KUKA KRL program: PROTON_EXHIBITION.src, PROTON_EXHIBITION.dat

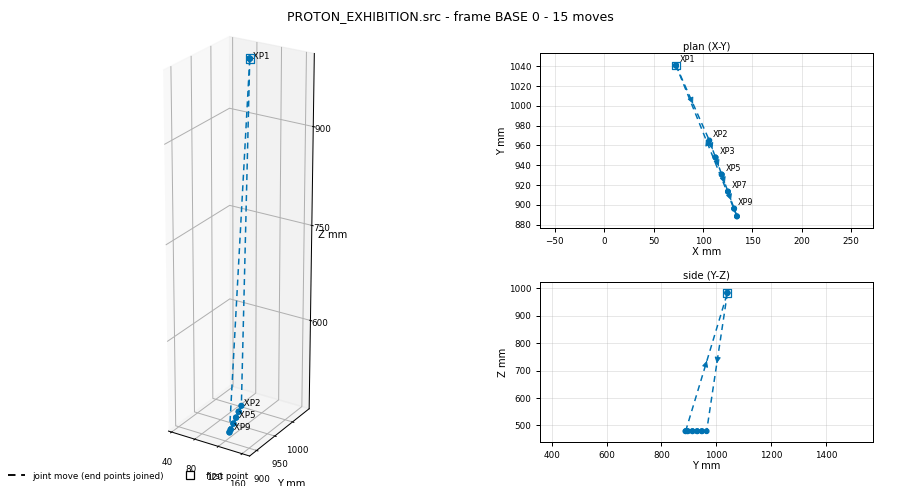
[picture p0: tool path of PROTON_EXHIBITION.src in frame BASE 0, 15 of 15 moves have a stored position in this frame; points joined in program order, loops and branches not executed]
--- PROTON_EXHIBITION.src ---
&ACCESS RVP
&REL 2
&PARAM DISKPATH = KRC:\\R1\\Program
DEF PROTON_EXHIBITION()
   DECL INT RET
   DECL INT CMD
   DECL REAL OUT_PULSE_TIME

   BAS(#INITMOV, 0)
   CMD = 0
   OUT_PULSE_TIME = 1.0

   \
       ;FOLD SPTP P1 Vel=100 % PDAT1 Tool[1]:Tool Base[0] ;%{PE}
       ;FOLD Parameters ;%{h}
       ;Params IlfProvider=kukaroboter.basistech.inlineforms.movement.spline; Kuka.IsGlobalPoint=False; Kuka.PointName=P1; Kuka.BlendingEnabled=False; Kuka.MoveDataPtpName=PDAT1; Kuka.VelocityPtp=100; Kuka.VelocityFieldEnabled=True; Kuka.ColDetectFieldEnabled=True; Kuka.CurrentCDSetIndex=0; Kuka.MovementParameterFieldEnabled=True; IlfCommand=SPTP
       ;ENDFOLD
       SPTP XP1 WITH $VEL_AXIS[1] = SVEL_JOINT(100.0), $TOOL = STOOL2(FP1), $BASE = SBASE(FP1.BASE_NO), $IPO_MODE = SIPO_MODE(FP1.IPO_FRAME), $LOAD = SLOAD(FP1.TOOL_NO), $ACC_AXIS[1] = SACC_JOINT(PPDAT1), $APO = SAPO_PTP(PPDAT1), $GEAR_JERK[1] = SGEAR_JERK(PPDAT1), $COLLMON_TOL_PRO[1] = USE_CM_PRO_VALUES(0)
       ;ENDFOLD

   LOOP
      ; ready to start = 0
      RET = EKI_SetInt("STATUS_EKI", "Status", 0)
      RET = EKI_Send("STATUS_EKI")

      ; wait for start cycle command, expected Cmd = 1
      CMD = 0
      REPEAT
         WAIT SEC 0.05
         RET = EKI_ReadNext("STATUS_EKI")
         IF RET == EkiOk THEN
            RET = EKI_GetInt("STATUS_EKI", "Cmd", CMD)
         ENDIF
      UNTIL (RET == EkiOk) AND (CMD == 1)

      ; next_position = 1
      RET = EKI_SetInt("STATUS_EKI", "Status", 1)
      RET = EKI_Send("STATUS_EKI")

   \
       ;FOLD SPTP P1 Vel=100 % PDAT1 Tool[1]:Tool Base[0] ;%{PE}
       ;FOLD Parameters ;%{h}
       ;Params IlfProvider=kukaroboter.basistech.inlineforms.movement.spline; Kuka.IsGlobalPoint=False; Kuka.PointName=P1; Kuka.BlendingEnabled=False; Kuka.MoveDataPtpName=PDAT1; Kuka.VelocityPtp=100; Kuka.VelocityFieldEnabled=True; Kuka.ColDetectFieldEnabled=True; Kuka.CurrentCDSetIndex=0; Kuka.MovementParameterFieldEnabled=True; IlfCommand=SPTP
       ;ENDFOLD
       SPTP XP1 WITH $VEL_AXIS[1] = SVEL_JOINT(100.0), $TOOL = STOOL2(FP1), $BASE = SBASE(FP1.BASE_NO), $IPO_MODE = SIPO_MODE(FP1.IPO_FRAME), $LOAD = SLOAD(FP1.TOOL_NO), $ACC_AXIS[1] = SACC_JOINT(PPDAT1), $APO = SAPO_PTP(PPDAT1), $GEAR_JERK[1] = SGEAR_JERK(PPDAT1), $COLLMON_TOL_PRO[1] = USE_CM_PRO_VALUES(0)
       ;ENDFOLD

      ; in_position = 2
      WAIT FOR $OUT[1] == FALSE
      RET = EKI_SetInt("STATUS_EKI", "Status", 2)
      RET = EKI_Send("STATUS_EKI")

      ; wait command to move to P2
      CMD = 0
      REPEAT
         WAIT SEC 0.05
         RET = EKI_ReadNext("STATUS_EKI")
         IF RET == EkiOk THEN
            RET = EKI_GetInt("STATUS_EKI", "Cmd", CMD)
         ENDIF
      UNTIL (RET == EkiOk) AND (CMD == 1)

      ; next_position = 1
      RET = EKI_SetInt("STATUS_EKI", "Status", 1)
      RET = EKI_Send("STATUS_EKI")
      PULSE($OUT[1], TRUE, OUT_PULSE_TIME)

      \
          ;FOLD SPTP P2 Vel=100 % PDAT2 Tool[1]:Tool Base[0] ;%{PE}
          ;FOLD Parameters ;%{h}
          ;Params IlfProvider=kukaroboter.basistech.inlineforms.movement.spline; Kuka.IsGlobalPoint=False; Kuka.PointName=P2; Kuka.BlendingEnabled=False; Kuka.MoveDataPtpName=PDAT2; Kuka.VelocityPtp=100; Kuka.VelocityFieldEnabled=True; Kuka.ColDetectFieldEnabled=True; Kuka.CurrentCDSetIndex=0; Kuka.MovementParameterFieldEnabled=True; IlfCommand=SPTP
          ;ENDFOLD
          SPTP XP2 WITH $VEL_AXIS[1] = SVEL_JOINT(100.0), $TOOL = STOOL2(FP2), $BASE = SBASE(FP2.BASE_NO), $IPO_MODE = SIPO_MODE(FP2.IPO_FRAME), $LOAD = SLOAD(FP2.TOOL_NO), $ACC_AXIS[1] = SACC_JOINT(PPDAT2), $APO = SAPO_PTP(PPDAT2), $GEAR_JERK[1] = SGEAR_JERK(PPDAT2), $COLLMON_TOL_PRO[1] = USE_CM_PRO_VALUES(0)
          ;ENDFOLD

      ; in_position = 2
      WAIT FOR $OUT[1] == FALSE
      RET = EKI_SetInt("STATUS_EKI", "Status", 2)
      RET = EKI_Send("STATUS_EKI")

      ; wait command to move to P3
      CMD = 0
      REPEAT
         WAIT SEC 0.05
         RET = EKI_ReadNext("STATUS_EKI")
         IF RET == EkiOk THEN
            RET = EKI_GetInt("STATUS_EKI", "Cmd", CMD)
         ENDIF
      UNTIL (RET == EkiOk) AND (CMD == 1)

      ; next_position = 1
      RET = EKI_SetInt("STATUS_EKI", "Status", 1)
      RET = EKI_Send("STATUS_EKI")
      PULSE($OUT[1], TRUE, OUT_PULSE_TIME)

      \
          ;FOLD SPTP P3 Vel=100 % PDAT3 Tool[1]:Tool Base[0] ;%{PE}
          ;FOLD Parameters ;%{h}
          ;Params IlfProvider=kukaroboter.basistech.inlineforms.movement.spline; Kuka.IsGlobalPoint=False; Kuka.PointName=P3; Kuka.BlendingEnabled=False; Kuka.MoveDataPtpName=PDAT3; Kuka.VelocityPtp=100; Kuka.VelocityFieldEnabled=True; Kuka.ColDetectFieldEnabled=True; Kuka.CurrentCDSetIndex=0; Kuka.MovementParameterFieldEnabled=True; IlfCommand=SPTP
          ;ENDFOLD
          SPTP XP3 WITH $VEL_AXIS[1] = SVEL_JOINT(100.0), $TOOL = STOOL2(FP3), $BASE = SBASE(FP3.BASE_NO), $IPO_MODE = SIPO_MODE(FP3.IPO_FRAME), $LOAD = SLOAD(FP3.TOOL_NO), $ACC_AXIS[1] = SACC_JOINT(PPDAT3), $APO = SAPO_PTP(PPDAT3), $GEAR_JERK[1] = SGEAR_JERK(PPDAT3), $COLLMON_TOL_PRO[1] = USE_CM_PRO_VALUES(0)
          ;ENDFOLD

      ; in_position = 2
      WAIT FOR $OUT[1] == FALSE
      RET = EKI_SetInt("STATUS_EKI", "Status", 2)
      RET = EKI_Send("STATUS_EKI")

      ; wait command to move to P4
      CMD = 0
      REPEAT
         WAIT SEC 0.05
         RET = EKI_ReadNext("STATUS_EKI")
         IF RET == EkiOk THEN
            RET = EKI_GetInt("STATUS_EKI", "Cmd", CMD)
         ENDIF
      UNTIL (RET == EkiOk) AND (CMD == 1)

      ; next_position = 1
      RET = EKI_SetInt("STATUS_EKI", "Status", 1)
      RET = EKI_Send("STATUS_EKI")
      PULSE($OUT[1], TRUE, OUT_PULSE_TIME)

      \
          ;FOLD SPTP P4 Vel=100 % PDAT4 Tool[1]:Tool Base[0] ;%{PE}
          ;FOLD Parameters ;%{h}
          ;Params IlfProvider=kukaroboter.basistech.inlineforms.movement.spline; Kuka.IsGlobalPoint=False; Kuka.PointName=P4; Kuka.BlendingEnabled=False; Kuka.MoveDataPtpName=PDAT4; Kuka.VelocityPtp=100; Kuka.VelocityFieldEnabled=True; Kuka.ColDetectFieldEnabled=True; Kuka.CurrentCDSetIndex=0; Kuka.MovementParameterFieldEnabled=True; IlfCommand=SPTP
          ;ENDFOLD
          SPTP XP4 WITH $VEL_AXIS[1] = SVEL_JOINT(100.0), $TOOL = STOOL2(FP4), $BASE = SBASE(FP4.BASE_NO), $IPO_MODE = SIPO_MODE(FP4.IPO_FRAME), $LOAD = SLOAD(FP4.TOOL_NO), $ACC_AXIS[1] = SACC_JOINT(PPDAT4), $APO = SAPO_PTP(PPDAT4), $GEAR_JERK[1] = SGEAR_JERK(PPDAT4), $COLLMON_TOL_PRO[1] = USE_CM_PRO_VALUES(0)
          ;ENDFOLD

      ; in_position = 2
      WAIT FOR $OUT[1] == FALSE
      RET = EKI_SetInt("STATUS_EKI", "Status", 2)
      RET = EKI_Send("STATUS_EKI")

      ; wait command to move to P5
      CMD = 0
      REPEAT
         WAIT SEC 0.05
         RET = EKI_ReadNext("STATUS_EKI")
         IF RET == EkiOk THEN
            RET = EKI_GetInt("STATUS_EKI", "Cmd", CMD)
         ENDIF
      UNTIL (RET == EkiOk) AND (CMD == 1)

      ; next_position = 1
      RET = EKI_SetInt("STATUS_EKI", "Status", 1)
      RET = EKI_Send("STATUS_EKI")
      PULSE($OUT[1], TRUE, OUT_PULSE_TIME)

      \
          ;FOLD SPTP P5 Vel=100 % PDAT5 Tool[1]:Tool Base[0] ;%{PE}
          ;FOLD Parameters ;%{h}
          ;Params IlfProvider=kukaroboter.basistech.inlineforms.movement.spline; Kuka.IsGlobalPoint=False; Kuka.PointName=P5; Kuka.BlendingEnabled=False; Kuka.MoveDataPtpName=PDAT5; Kuka.VelocityPtp=100; Kuka.VelocityFieldEnabled=True; Kuka.ColDetectFieldEnabled=True; Kuka.CurrentCDSetIndex=0; Kuka.MovementParameterFieldEnabled=True; IlfCommand=SPTP
          ;ENDFOLD
          SPTP XP5 WITH $VEL_AXIS[1] = SVEL_JOINT(100.0), $TOOL = STOOL2(FP5), $BASE = SBASE(FP5.BASE_NO), $IPO_MODE = SIPO_MODE(FP5.IPO_FRAME), $LOAD = SLOAD(FP5.TOOL_NO), $ACC_AXIS[1] = SACC_JOINT(PPDAT5), $APO = SAPO_PTP(PPDAT5), $GEAR_JERK[1] = SGEAR_JERK(PPDAT5), $COLLMON_TOL_PRO[1] = USE_CM_PRO_VALUES(0)
          ;ENDFOLD

      ; in_position = 2
      WAIT FOR $OUT[1] == FALSE
      RET = EKI_SetInt("STATUS_EKI", "Status", 2)
      RET = EKI_Send("STATUS_EKI")

      ; wait command to move to P6
      CMD = 0
      REPEAT
         WAIT SEC 0.05
         RET = EKI_ReadNext("STATUS_EKI")
         IF RET == EkiOk THEN
            RET = EKI_GetInt("STATUS_EKI", "Cmd", CMD)
         ENDIF
      UNTIL (RET == EkiOk) AND (CMD == 1)

      ; next_position = 1
      RET = EKI_SetInt("STATUS_EKI", "Status", 1)
      RET = EKI_Send("STATUS_EKI")
      PULSE($OUT[1], TRUE, OUT_PULSE_TIME)

      \
          ;FOLD SPTP P6 Vel=100 % PDAT6 Tool[1]:Tool Base[0] ;%{PE}
          ;FOLD Parameters ;%{h}
          ;Params IlfProvider=kukaroboter.basistech.inlineforms.movement.spline; Kuka.IsGlobalPoint=False; Kuka.PointName=P6; Kuka.BlendingEnabled=False; Kuka.MoveDataPtpName=PDAT6; Kuka.VelocityPtp=100; Kuka.VelocityFieldEnabled=True; Kuka.ColDetectFieldEnabled=True; Kuka.CurrentCDSetIndex=0; Kuka.MovementParameterFieldEnabled=True; IlfCommand=SPTP
          ;ENDFOLD
          SPTP XP6 WITH $VEL_AXIS[1] = SVEL_JOINT(100.0), $TOOL = STOOL2(FP6), $BASE = SBASE(FP6.BASE_NO), $IPO_MODE = SIPO_MODE(FP6.IPO_FRAME), $LOAD = SLOAD(FP6.TOOL_NO), $ACC_AXIS[1] = SACC_JOINT(PPDAT6), $APO = SAPO_PTP(PPDAT6), $GEAR_JERK[1] = SGEAR_JERK(PPDAT6), $COLLMON_TOL_PRO[1] = USE_CM_PRO_VALUES(0)
          ;ENDFOLD

      ; in_position = 2
      WAIT FOR $OUT[1] == FALSE
      RET = EKI_SetInt("STATUS_EKI", "Status", 2)
      RET = EKI_Send("STATUS_EKI")

      ; wait command to move to P7
      CMD = 0
      REPEAT
         WAIT SEC 0.05
         RET = EKI_ReadNext("STATUS_EKI")
         IF RET == EkiOk THEN
            RET = EKI_GetInt("STATUS_EKI", "Cmd", CMD)
         ENDIF
      UNTIL (RET == EkiOk) AND (CMD == 1)

      ; next_position = 1
      RET = EKI_SetInt("STATUS_EKI", "Status", 1)
      RET = EKI_Send("STATUS_EKI")
      PULSE($OUT[1], TRUE, OUT_PULSE_TIME)

      \
          ;FOLD SPTP P7 Vel=100 % PDAT7 Tool[1]:Tool Base[0] ;%{PE}
          ;FOLD Parameters ;%{h}
          ;Params IlfProvider=kukaroboter.basistech.inlineforms.movement.spline; Kuka.IsGlobalPoint=False; Kuka.PointName=P7; Kuka.BlendingEnabled=False; Kuka.MoveDataPtpName=PDAT7; Kuka.VelocityPtp=100; Kuka.VelocityFieldEnabled=True; Kuka.ColDetectFieldEnabled=True; Kuka.CurrentCDSetIndex=0; Kuka.MovementParameterFieldEnabled=True; IlfCommand=SPTP
          ;ENDFOLD
          SPTP XP7 WITH $VEL_AXIS[1] = SVEL_JOINT(100.0), $TOOL = STOOL2(FP7), $BASE = SBASE(FP7.BASE_NO), $IPO_MODE = SIPO_MODE(FP7.IPO_FRAME), $LOAD = SLOAD(FP7.TOOL_NO), $ACC_AXIS[1] = SACC_JOINT(PPDAT7), $APO = SAPO_PTP(PPDAT7), $GEAR_JERK[1] = SGEAR_JERK(PPDAT7), $COLLMON_TOL_PRO[1] = USE_CM_PRO_VALUES(0)
          ;ENDFOLD

      ; in_position = 2
      WAIT FOR $OUT[1] == FALSE
      RET = EKI_SetInt("STATUS_EKI", "Status", 2)
      RET = EKI_Send("STATUS_EKI")

      ; wait command to move to P8
      CMD = 0
      REPEAT
         WAIT SEC 0.05
         RET = EKI_ReadNext("STATUS_EKI")
         IF RET == EkiOk THEN
            RET = EKI_GetInt("STATUS_EKI", "Cmd", CMD)
         ENDIF
      UNTIL (RET == EkiOk) AND (CMD == 1)

      ; next_position = 1
      RET = EKI_SetInt("STATUS_EKI", "Status", 1)
      RET = EKI_Send("STATUS_EKI")
      PULSE($OUT[1], TRUE, OUT_PULSE_TIME)

      \
          ;FOLD SPTP P8 Vel=100 % PDAT8 Tool[1]:Tool Base[0] ;%{PE}
          ;FOLD Parameters ;%{h}
          ;Params IlfProvider=kukaroboter.basistech.inlineforms.movement.spline; Kuka.IsGlobalPoint=False; Kuka.PointName=P8; Kuka.BlendingEnabled=False; Kuka.MoveDataPtpName=PDAT8; Kuka.VelocityPtp=100; Kuka.VelocityFieldEnabled=True; Kuka.ColDetectFieldEnabled=True; Kuka.CurrentCDSetIndex=0; Kuka.MovementParameterFieldEnabled=True; IlfCommand=SPTP
          ;ENDFOLD
          SPTP XP8 WITH $VEL_AXIS[1] = SVEL_JOINT(100.0), $TOOL = STOOL2(FP8), $BASE = SBASE(FP8.BASE_NO), $IPO_MODE = SIPO_MODE(FP8.IPO_FRAME), $LOAD = SLOAD(FP8.TOOL_NO), $ACC_AXIS[1] = SACC_JOINT(PPDAT8), $APO = SAPO_PTP(PPDAT8), $GEAR_JERK[1] = SGEAR_JERK(PPDAT8), $COLLMON_TOL_PRO[1] = USE_CM_PRO_VALUES(0)
          ;ENDFOLD

      ; in_position = 2
      WAIT FOR $OUT[1] == FALSE
      RET = EKI_SetInt("STATUS_EKI", "Status", 2)
      RET = EKI_Send("STATUS_EKI")

      ; wait command to move to P9
      CMD = 0
      REPEAT
         WAIT SEC 0.05
         RET = EKI_ReadNext("STATUS_EKI")
         IF RET == EkiOk THEN
            RET = EKI_GetInt("STATUS_EKI", "Cmd", CMD)
         ENDIF
      UNTIL (RET == EkiOk) AND (CMD == 1)

      ; next_position = 1
      RET = EKI_SetInt("STATUS_EKI", "Status", 1)
      RET = EKI_Send("STATUS_EKI")
      PULSE($OUT[1], TRUE, OUT_PULSE_TIME)

      \
          ;FOLD SPTP P9 Vel=100 % PDAT9 Tool[1]:Tool Base[0] ;%{PE}
          ;FOLD Parameters ;%{h}
          ;Params IlfProvider=kukaroboter.basistech.inlineforms.movement.spline; Kuka.IsGlobalPoint=False; Kuka.PointName=P9; Kuka.BlendingEnabled=False; Kuka.MoveDataPtpName=PDAT9; Kuka.VelocityPtp=100; Kuka.VelocityFieldEnabled=True; Kuka.ColDetectFieldEnabled=True; Kuka.CurrentCDSetIndex=0; Kuka.MovementParameterFieldEnabled=True; IlfCommand=SPTP
          ;ENDFOLD
          SPTP XP9 WITH $VEL_AXIS[1] = SVEL_JOINT(100.0), $TOOL = STOOL2(FP9), $BASE = SBASE(FP9.BASE_NO), $IPO_MODE = SIPO_MODE(FP9.IPO_FRAME), $LOAD = SLOAD(FP9.TOOL_NO), $ACC_AXIS[1] = SACC_JOINT(PPDAT9), $APO = SAPO_PTP(PPDAT9), $GEAR_JERK[1] = SGEAR_JERK(PPDAT9), $COLLMON_TOL_PRO[1] = USE_CM_PRO_VALUES(0)
          ;ENDFOLD

      ; in_position = 2
      WAIT FOR $OUT[1] == FALSE
      RET = EKI_SetInt("STATUS_EKI", "Status", 2)
      RET = EKI_Send("STATUS_EKI")

      ; wait command to move to P10
      CMD = 0
      REPEAT
         WAIT SEC 0.05
         RET = EKI_ReadNext("STATUS_EKI")
         IF RET == EkiOk THEN
            RET = EKI_GetInt("STATUS_EKI", "Cmd", CMD)
         ENDIF
      UNTIL (RET == EkiOk) AND (CMD == 1)

      ; next_position = 1
      RET = EKI_SetInt("STATUS_EKI", "Status", 1)
      RET = EKI_Send("STATUS_EKI")
      PULSE($OUT[1], TRUE, OUT_PULSE_TIME)

      \
          ;FOLD SPTP P10 Vel=100 % PDAT10 Tool[1]:Tool Base[0] ;%{PE}
          ;FOLD Parameters ;%{h}
          ;Params IlfProvider=kukaroboter.basistech.inlineforms.movement.spline; Kuka.IsGlobalPoint=False; Kuka.PointName=P10; Kuka.BlendingEnabled=False; Kuka.MoveDataPtpName=PDAT10; Kuka.VelocityPtp=100; Kuka.VelocityFieldEnabled=True; Kuka.ColDetectFieldEnabled=True; Kuka.CurrentCDSetIndex=0; Kuka.MovementParameterFieldEnabled=True; IlfCommand=SPTP
          ;ENDFOLD
          SPTP XP10 WITH $VEL_AXIS[1] = SVEL_JOINT(100.0), $TOOL = STOOL2(FP10), $BASE = SBASE(FP10.BASE_NO), $IPO_MODE = SIPO_MODE(FP10.IPO_FRAME), $LOAD = SLOAD(FP10.TOOL_NO), $ACC_AXIS[1] = SACC_JOINT(PPDAT10), $APO = SAPO_PTP(PPDAT10), $GEAR_JERK[1] = SGEAR_JERK(PPDAT10), $COLLMON_TOL_PRO[1] = USE_CM_PRO_VALUES(0)
          ;ENDFOLD

      ; in_position = 2
      WAIT FOR $OUT[1] == FALSE
      RET = EKI_SetInt("STATUS_EKI", "Status", 2)
      RET = EKI_Send("STATUS_EKI")

      ; wait command to move to P11
      CMD = 0
      REPEAT
         WAIT SEC 0.05
         RET = EKI_ReadNext("STATUS_EKI")
         IF RET == EkiOk THEN
            RET = EKI_GetInt("STATUS_EKI", "Cmd", CMD)
         ENDIF
      UNTIL (RET == EkiOk) AND (CMD == 1)

      ; next_position = 1
      RET = EKI_SetInt("STATUS_EKI", "Status", 1)
      RET = EKI_Send("STATUS_EKI")
      PULSE($OUT[1], TRUE, OUT_PULSE_TIME)

      \
          ;FOLD SPTP P11 Vel=100 % PDAT11 Tool[1]:Tool Base[0] ;%{PE}
          ;FOLD Parameters ;%{h}
          ;Params IlfProvider=kukaroboter.basistech.inlineforms.movement.spline; Kuka.IsGlobalPoint=False; Kuka.PointName=P11; Kuka.BlendingEnabled=False; Kuka.MoveDataPtpName=PDAT11; Kuka.VelocityPtp=100; Kuka.VelocityFieldEnabled=True; Kuka.ColDetectFieldEnabled=True; Kuka.CurrentCDSetIndex=0; Kuka.MovementParameterFieldEnabled=True; IlfCommand=SPTP
          ;ENDFOLD
          SPTP XP11 WITH $VEL_AXIS[1] = SVEL_JOINT(100.0), $TOOL = STOOL2(FP11), $BASE = SBASE(FP11.BASE_NO), $IPO_MODE = SIPO_MODE(FP11.IPO_FRAME), $LOAD = SLOAD(FP11.TOOL_NO), $ACC_AXIS[1] = SACC_JOINT(PPDAT11), $APO = SAPO_PTP(PPDAT11), $GEAR_JERK[1] = SGEAR_JERK(PPDAT11), $COLLMON_TOL_PRO[1] = USE_CM_PRO_VALUES(0)
          ;ENDFOLD

      ; in_position = 2
      WAIT FOR $OUT[1] == FALSE
      RET = EKI_SetInt("STATUS_EKI", "Status", 2)
      RET = EKI_Send("STATUS_EKI")

      ; wait command to move to P12
      CMD = 0
      REPEAT
         WAIT SEC 0.05
         RET = EKI_ReadNext("STATUS_EKI")
         IF RET == EkiOk THEN
            RET = EKI_GetInt("STATUS_EKI", "Cmd", CMD)
         ENDIF
      UNTIL (RET == EkiOk) AND (CMD == 1)

      ; next_position = 1
      RET = EKI_SetInt("STATUS_EKI", "Status", 1)
      RET = EKI_Send("STATUS_EKI")
      PULSE($OUT[1], TRUE, OUT_PULSE_TIME)

      \
          ;FOLD SPTP P12 Vel=100 % PDAT12 Tool[1]:Tool Base[0] ;%{PE}
          ;FOLD Parameters ;%{h}
          ;Params IlfProvider=kukaroboter.basistech.inlineforms.movement.spline; Kuka.IsGlobalPoint=False; Kuka.PointName=P12; Kuka.BlendingEnabled=False; Kuka.MoveDataPtpName=PDAT12; Kuka.VelocityPtp=100; Kuka.VelocityFieldEnabled=True; Kuka.ColDetectFieldEnabled=True; Kuka.CurrentCDSetIndex=0; Kuka.MovementParameterFieldEnabled=True; IlfCommand=SPTP
          ;ENDFOLD
          SPTP XP12 WITH $VEL_AXIS[1] = SVEL_JOINT(100.0), $TOOL = STOOL2(FP12), $BASE = SBASE(FP12.BASE_NO), $IPO_MODE = SIPO_MODE(FP12.IPO_FRAME), $LOAD = SLOAD(FP12.TOOL_NO), $ACC_AXIS[1] = SACC_JOINT(PPDAT12), $APO = SAPO_PTP(PPDAT12), $GEAR_JERK[1] = SGEAR_JERK(PPDAT12), $COLLMON_TOL_PRO[1] = USE_CM_PRO_VALUES(0)
          ;ENDFOLD

      ; in_position = 2
      WAIT FOR $OUT[1] == FALSE
      RET = EKI_SetInt("STATUS_EKI", "Status", 2)
      RET = EKI_Send("STATUS_EKI")

      ; wait command to move to P13
      CMD = 0
      REPEAT
         WAIT SEC 0.05
         RET = EKI_ReadNext("STATUS_EKI")
         IF RET == EkiOk THEN
            RET = EKI_GetInt("STATUS_EKI", "Cmd", CMD)
         ENDIF
      UNTIL (RET == EkiOk) AND (CMD == 1)

      ; next_position = 1
      RET = EKI_SetInt("STATUS_EKI", "Status", 1)
      RET = EKI_Send("STATUS_EKI")
      PULSE($OUT[1], TRUE, OUT_PULSE_TIME)

      \
          ;FOLD SPTP P13 Vel=100 % PDAT13 Tool[1]:Tool Base[0] ;%{PE}
          ;FOLD Parameters ;%{h}
          ;Params IlfProvider=kukaroboter.basistech.inlineforms.movement.spline; Kuka.IsGlobalPoint=False; Kuka.PointName=P13; Kuka.BlendingEnabled=False; Kuka.MoveDataPtpName=PDAT13; Kuka.VelocityPtp=100; Kuka.VelocityFieldEnabled=True; Kuka.ColDetectFieldEnabled=True; Kuka.CurrentCDSetIndex=0; Kuka.MovementParameterFieldEnabled=True; IlfCommand=SPTP
          ;ENDFOLD
          SPTP XP13 WITH $VEL_AXIS[1] = SVEL_JOINT(100.0), $TOOL = STOOL2(FP13), $BASE = SBASE(FP13.BASE_NO), $IPO_MODE = SIPO_MODE(FP13.IPO_FRAME), $LOAD = SLOAD(FP13.TOOL_NO), $ACC_AXIS[1] = SACC_JOINT(PPDAT13), $APO = SAPO_PTP(PPDAT13), $GEAR_JERK[1] = SGEAR_JERK(PPDAT13), $COLLMON_TOL_PRO[1] = USE_CM_PRO_VALUES(0)
          ;ENDFOLD

      ; in_position = 2
      WAIT FOR $OUT[1] == FALSE
      RET = EKI_SetInt("STATUS_EKI", "Status", 2)
      RET = EKI_Send("STATUS_EKI")

      ; wait command to return to P1
      CMD = 0
      REPEAT
         WAIT SEC 0.05
         RET = EKI_ReadNext("STATUS_EKI")
         IF RET == EkiOk THEN
            RET = EKI_GetInt("STATUS_EKI", "Cmd", CMD)
         ENDIF
      UNTIL (RET == EkiOk) AND (CMD == 1)

      ; next_position = 1
      RET = EKI_SetInt("STATUS_EKI", "Status", 1)
      RET = EKI_Send("STATUS_EKI")

      \
          ;FOLD SPTP P1 Vel=100 % PDAT1 Tool[1]:Tool Base[0] ;%{PE}
          ;FOLD Parameters ;%{h}
          ;Params IlfProvider=kukaroboter.basistech.inlineforms.movement.spline; Kuka.IsGlobalPoint=False; Kuka.PointName=P1; Kuka.BlendingEnabled=False; Kuka.MoveDataPtpName=PDAT1; Kuka.VelocityPtp=100; Kuka.VelocityFieldEnabled=True; Kuka.ColDetectFieldEnabled=True; Kuka.CurrentCDSetIndex=0; Kuka.MovementParameterFieldEnabled=True; IlfCommand=SPTP
          ;ENDFOLD
          SPTP XP1 WITH $VEL_AXIS[1] = SVEL_JOINT(100.0), $TOOL = STOOL2(FP1), $BASE = SBASE(FP1.BASE_NO), $IPO_MODE = SIPO_MODE(FP1.IPO_FRAME), $LOAD = SLOAD(FP1.TOOL_NO), $ACC_AXIS[1] = SACC_JOINT(PPDAT1), $APO = SAPO_PTP(PPDAT1), $GEAR_JERK[1] = SGEAR_JERK(PPDAT1), $COLLMON_TOL_PRO[1] = USE_CM_PRO_VALUES(0)
          ;ENDFOLD

      ; back to first position, ready to start = 0
      RET = EKI_SetInt("STATUS_EKI", "Status", 0)
      RET = EKI_Send("STATUS_EKI")

   ENDLOOP
END

--- PROTON_EXHIBITION.dat ---
&ACCESS RVP
&REL 2
&PARAM DISKPATH = KRC:\\R1\\Program
DEFDAT  PROTON_EXHIBITION
;FOLD EXTERNAL DECLARATIONS;%{PE}%MKUKATPBASIS,%CEXT,%VCOMMON,%P
;FOLD BASISTECH EXT;%{PE}%MKUKATPBASIS,%CEXT,%VEXT,%P
EXT  BAS (BAS_COMMAND  :IN,REAL  :IN )
DECL INT SUCCESS
;ENDFOLD (BASISTECH EXT)
;FOLD USER EXT;%{E}%MKUKATPUSER,%CEXT,%VEXT,%P
;Make your modifications here

;ENDFOLD (USER EXT)
;ENDFOLD (EXTERNAL DECLARATIONS)
DECL E6POS XP1={ X 72.744058, Y 1040.860681, Z 983.603439, A -160.000000, B 0.000051, C 90.000000, S 22, T 19, E1 0.0, E2 0.0, E3 0.0, E4 0.0, E5 0.0, E6 0.0 }
DECL FDAT FP1 = { BASE_NO 0, TOOL_NO 1, IPO_FRAME #BASE, POINT2[] " " }
DECL PDAT PPDAT1={ACC 100.000,APO_DIST 500.000,APO_MODE #CDIS,GEAR_JERK 100.000,EXAX_IGN 0}
DECL E6POS XP2={ X 106.398535, Y 965.069035, Z 479.071032, A -160.000018, B 0.000056, C 134.999980, S 22, T 19, E1 0.0, E2 0.0, E3 0.0, E4 0.0, E5 0.0, E6 0.0 }
DECL FDAT FP2 = { BASE_NO 0, TOOL_NO 1, IPO_FRAME #BASE, POINT2[] " " }
DECL PDAT PPDAT2={ACC 100.000,APO_DIST 500.000,APO_MODE #CDIS,GEAR_JERK 100.000,EXAX_IGN 0}
DECL E6POS XP3={ X 112.668856, Y 947.841308, Z 479.070952, A -160.000015, B 0.000050, C 119.999992, S 22, T 19, E1 0.0, E2 0.0, E3 0.0, E4 0.0, E5 0.0, E6 0.0 }
DECL FDAT FP3 = { BASE_NO 0, TOOL_NO 1, IPO_FRAME #BASE, POINT2[] " " }
DECL PDAT PPDAT3={ACC 100.000,APO_DIST 500.000,APO_MODE #CDIS,GEAR_JERK 100.000,EXAX_IGN 0}
DECL E6POS XP4={ X 112.668856, Y 947.841308, Z 479.070952, A -160.000015, B 0.000050, C 119.999992, S 22, T 19, E1 0.0, E2 0.0, E3 0.0, E4 0.0, E5 0.0, E6 0.0 }
DECL FDAT FP4 = { BASE_NO 0, TOOL_NO 1, IPO_FRAME #BASE, POINT2[] " " }
DECL PDAT PPDAT4={ACC 100.000,APO_DIST 500.000,APO_MODE #CDIS,GEAR_JERK 100.000,EXAX_IGN 0}
DECL E6POS XP5={ X 118.939200, Y 930.613562, Z 479.070894, A 19.999984, B -0.000057, C -104.999996, S 22, T 19, E1 0.0, E2 0.0, E3 0.0, E4 0.0, E5 0.0, E6 0.0 }
DECL FDAT FP5 = { BASE_NO 0, TOOL_NO 1, IPO_FRAME #BASE, POINT2[] " " }
DECL PDAT PPDAT5={ACC 100.000,APO_DIST 500.000,APO_MODE #CDIS,GEAR_JERK 100.000,EXAX_IGN 0}
DECL E6POS XP6={ X 118.939200, Y 930.613562, Z 479.070894, A 19.999984, B -0.000057, C -104.999996, S 22, T 19, E1 0.0, E2 0.0, E3 0.0, E4 0.0, E5 0.0, E6 0.0 }
DECL FDAT FP6 = { BASE_NO 0, TOOL_NO 1, IPO_FRAME #BASE, POINT2[] " " }
DECL PDAT PPDAT6={ACC 100.000,APO_DIST 500.000,APO_MODE #CDIS,GEAR_JERK 100.000,EXAX_IGN 0}
DECL E6POS XP7={ X 125.209589, Y 913.385922, Z 479.070942, A 19.999960, B -0.000044, C -90.000001, S 22, T 19, E1 0.0, E2 0.0, E3 0.0, E4 0.0, E5 0.0, E6 0.0 }
DECL FDAT FP7 = { BASE_NO 0, TOOL_NO 1, IPO_FRAME #BASE, POINT2[] " " }
DECL PDAT PPDAT7={ACC 100.000,APO_DIST 500.000,APO_MODE #CDIS,GEAR_JERK 100.000,EXAX_IGN 0}
DECL E6POS XP8={ X 125.209589, Y 913.385922, Z 479.070942, A 19.999960, B -0.000044, C -90.000001, S 22, T 19, E1 0.0, E2 0.0, E3 0.0, E4 0.0, E5 0.0, E6 0.0 }
DECL FDAT FP8 = { BASE_NO 0, TOOL_NO 1, IPO_FRAME #BASE, POINT2[] " " }
DECL PDAT PPDAT8={ACC 100.000,APO_DIST 500.000,APO_MODE #CDIS,GEAR_JERK 100.000,EXAX_IGN 0}
DECL E6POS XP9={ X 131.480033, Y 896.158220, Z 479.070968, A 19.999973, B -0.000043, C -74.999983, S 22, T 19, E1 0.0, E2 0.0, E3 0.0, E4 0.0, E5 0.0, E6 0.0 }
DECL FDAT FP9 = { BASE_NO 0, TOOL_NO 1, IPO_FRAME #BASE, POINT2[] " " }
DECL PDAT PPDAT9={ACC 100.000,APO_DIST 500.000,APO_MODE #CDIS,GEAR_JERK 100.000,EXAX_IGN 0}
DECL E6POS XP10={ X 131.480033, Y 896.158220, Z 479.070968, A 19.999973, B -0.000043, C -74.999983, S 22, T 19, E1 0.0, E2 0.0, E3 0.0, E4 0.0, E5 0.0, E6 0.0 }
DECL FDAT FP10 = { BASE_NO 0, TOOL_NO 1, IPO_FRAME #BASE, POINT2[] " " }
DECL PDAT PPDAT10={ACC 100.000,APO_DIST 500.000,APO_MODE #CDIS,GEAR_JERK 100.000,EXAX_IGN 0}
DECL E6POS XP11={ X 134.330152, Y 888.327419, Z 479.071105, A 19.999986, B -0.000028, C -59.999982, S 22, T 19, E1 0.0, E2 0.0, E3 0.0, E4 0.0, E5 0.0, E6 0.0 }
DECL FDAT FP11 = { BASE_NO 0, TOOL_NO 1, IPO_FRAME #BASE, POINT2[] " " }
DECL PDAT PPDAT11={ACC 100.000,APO_DIST 500.000,APO_MODE #CDIS,GEAR_JERK 100.000,EXAX_IGN 0}
DECL E6POS XP12={ X 134.330152, Y 888.327419, Z 479.071105, A 19.999986, B -0.000028, C -59.999982, S 22, T 19, E1 0.0, E2 0.0, E3 0.0, E4 0.0, E5 0.0, E6 0.0 }
DECL FDAT FP12 = { BASE_NO 0, TOOL_NO 1, IPO_FRAME #BASE, POINT2[] " " }
DECL PDAT PPDAT12={ACC 100.000,APO_DIST 500.000,APO_MODE #CDIS,GEAR_JERK 100.000,EXAX_IGN 0}
DECL E6POS XP13={ X 72.744058, Y 1040.860681, Z 983.603439, A -160.000000, B 0.000051, C 90.000000, S 22, T 19, E1 0.0, E2 0.0, E3 0.0, E4 0.0, E5 0.0, E6 0.0 }
DECL FDAT FP13 = { BASE_NO 0, TOOL_NO 1, IPO_FRAME #BASE, POINT2[] " " }
DECL PDAT PPDAT13={ACC 100.000,APO_DIST 500.000,APO_MODE #CDIS,GEAR_JERK 100.000,EXAX_IGN 0}
ENDDAT
